{attribute 'qualified_only'}
VAR_GLOBAL

	
END_VAR

(* stored: Version 1.1.0.1, ProductVersion 3.1.4024.3
   GVL Control: Id {3ea5403b-0fbe-4b19-8f13-45713f688109} *)
